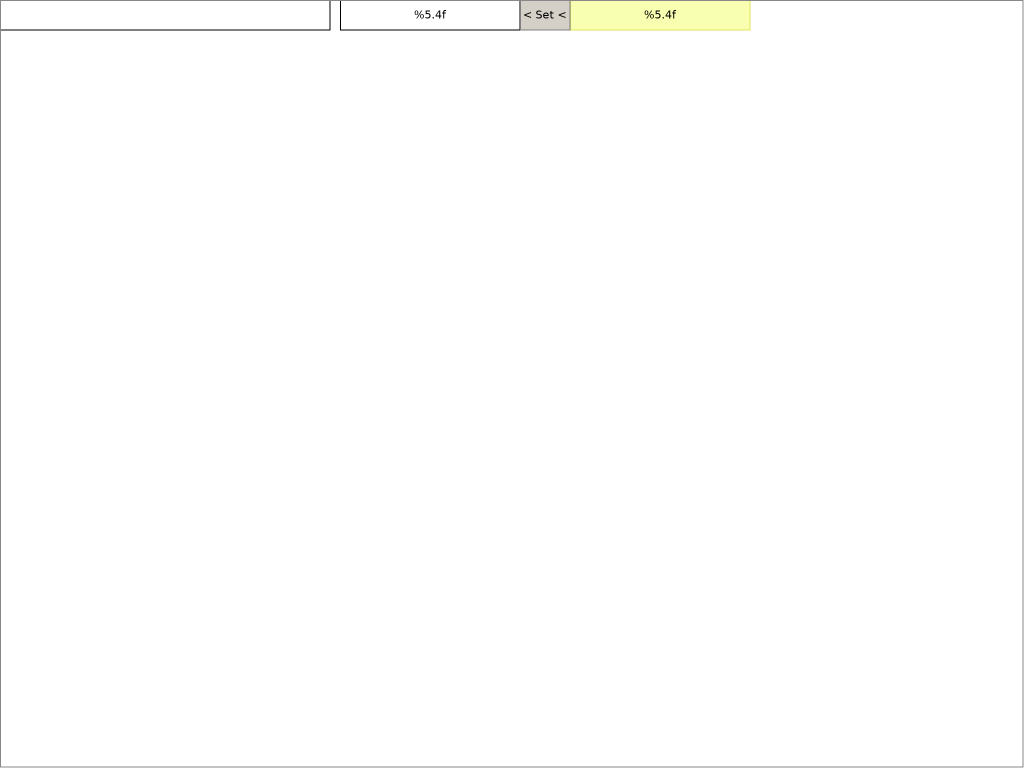
VISUALIZATION Param_LREAL_Supply  // 1024x768
VAR_INPUT
	nIdx:		INT;
END_VAR
    Rectangle (340,0 180x30), "%5.4f", text variable: stSupply_Visu.fLrealAktValue[nIdx]
    Rectangle (0,0 330x30), text list: 'TL_Supply', text index: nIdx
    Rectangle (570,0 180x30), "%5.4f", text variable: stSupply_Visu.fLrealNewValue[nIdx]
        OnMouseClick: write the text variable via Default
    Rectangle (520,0 50x30), "< Set <"
        OnMouseClick: execute { stSupply_Visu.bLrealSetValue[nIdx]:=TRUE; }
END_VISUALIZATION

(* stored: Version 1.1.0.1
   Visu Param_LREAL_Supply: Id {1e83c250-1412-4113-b72a-1860a1442b8b} *)
